(* Schneider Machine Expert - Basic project memorywords, file version 1.9.0.0 *)
(* ProjectInformations: Name=New project *)

HARDWARE
  Cpu 0: TM221CE16R
  EthernetConfiguration: NetworkName=M221, IpAllocationMode=FixedAddress, IpAddress=0.0.0.0, SubnetMask=0.0.0.0
  SerialLineConfiguration: Baud=Baud19200, Parity=ParityEven, DataBits=DataBits8, StopBits=StopBits1, PhysicalMedium=PhysicalMediumRs485, TransmissionMode=TransmissionModeModbusRtu, SlaveId=1, Addressing=SlaveAddressing
  MastTask: UsePeriodScanMode=false, PeriodScan=100
  FastTask: Period=255
  CpuBehavior: StartingMode=StartAsPreviousState, AutoSaveRamOnEeprom=true, WatchdogPeriod=250

SYMBOLS  (address, symbol, comment, settings)

POU New POU
  (* SectionNumber=1 *)

// Rung 0
  LD %I0.0
  [ %MW107 := (%mw1 +1) * 2 ]
  // as ST:
  //   IF %I0.0 THEN %MW107 := (%mw1 +1) * 2; END_IF;

// Rung 1
  LD 1
  [ %MW1 := 2 ]
  // as ST:
  //   %MW1 := 2;
